FUNCTION_BLOCK FB_Lifter
VAR_OUTPUT
	bLifter: BOOL;
	bImukuppi: BOOL;
END_VAR
VAR
	DelayStart: BOOL;
	tonImukuppiDelay: TON := (PT := TIME#2s0ms);
	LifterState: E_LifterState;
	NostoCMD: BOOL;
	bKplKyydissa: BOOL;
	LaskuCMD: BOOL;
END_VAR
VAR_OUTPUT
	Ready: BOOL;
END_VAR


tonImukuppiDelay(IN := DelayStart);



CASE LifterState OF
	
	E_LifterState.KplEiKyydissa:
		Ready := TRUE;
		IF NostoCMD = TRUE THEN
			LifterState := E_LifterState.NostoAlas;
			Ready := FALSE;
		END_IF
	
	E_LifterState.NostoAlas:
		Ready := FALSE;
		bLifter := TRUE;
		tonImukuppiDelay.PT := T#1S;
		DelayStart := TRUE;
		IF tonImukuppiDelay.Q THEN
			DelayStart := FALSE;
			LifterState := E_LifterState.NostoImukuppi;
		END_IF
	
	E_LifterState.NostoImukuppi:
		bImukuppi := TRUE;
		bLifter := TRUE;
		tonImukuppiDelay.PT := T#2S;
		DelayStart := TRUE;
		IF tonImukuppiDelay.Q THEN
			DelayStart := FALSE;
			LifterState := E_LifterState.NostoYlos;
		END_IF
	
	E_LifterState.NostoYlos:
		bLifter := FALSE;
		tonImukuppiDelay.PT := T#2S;
		DelayStart := TRUE;
		IF tonImukuppiDelay.Q THEN
			DelayStart := FALSE;
			LifterState := E_LifterState.KplKyydissa;
		END_IF	
	
	/////////////////////
	
	E_LifterState.KplKyydissa:
		Ready := TRUE;
		bKplKyydissa :=TRUE;
		IF LaskuCMD = TRUE THEN
			Ready := FALSE;
			LifterState := E_LifterState.LaskuAlas;
		END_IF
	
	/////////////////////////
	
	
	E_LifterState.LaskuAlas:
		Ready := FALSE;
		bLifter := TRUE;
		tonImukuppiDelay.PT := T#1S;
		DelayStart := TRUE;
		IF tonImukuppiDelay.Q THEN
			DelayStart := FALSE;
			LifterState := E_LifterState.LaskuImukuppi;
		END_IF
	
	E_LifterState.LaskuImukuppi:
		bImukuppi := FALSE;
		bLifter := TRUE;
		tonImukuppiDelay.PT := T#2S;
		DelayStart := TRUE;
		IF tonImukuppiDelay.Q THEN
			DelayStart := FALSE;
			LifterState := E_LifterState.LaskuYlos;
		END_IF
	
	E_LifterState.LaskuYlos:
		bLifter := FALSE;
		tonImukuppiDelay.PT := T#2S;
		DelayStart := TRUE;
		IF tonImukuppiDelay.Q THEN
			DelayStart := FALSE;
			LifterState := E_LifterState.KplEiKyydissa;
		END_IF	
	
END_CASE

LaskuCMD := FALSE;
NostoCMD := FALSE;

METHOD KplLasku : BOOL
VAR_INPUT
END_VAR
LaskuCMD := TRUE;
END_METHOD

METHOD KplNosto : BOOL
NostoCMD := TRUE;
END_METHOD

END_FUNCTION_BLOCK

(* stored: Version 1.1.0.1, ProductVersion 3.1.4024.12
   POU FB_Lifter: Id {5783411b-d6ff-44ed-8a5b-d08f1ab0363a}, SpecialFunc None
   Method KplLasku: Id {2ea166f5-e773-407e-a6ba-55ba8b8a5ad5}
   Method KplNosto: Id {7747a54a-c261-4a6a-84d9-63b8b0585b6f} *)
